// TIA Portal V17 export
// export: Created 2024-09-02T12:50:26.1404995Z, ExportSetting WithDefaults, DisplayName Totally Integrated Automation Portal, DisplayVersion V17, DisplayName TIA Portal Openness, DisplayVersion V17, DisplayName TIA Portal Version Control Interface, DisplayVersion V17, DisplayName STEP 7 Professional, DisplayVersion V17, DisplayName STEP 7 Safety, DisplayVersion V17, DisplayName WinCC Professional, DisplayVersion V17
TYPE "type_HMI_EKS_DATA"
// stored: IsFailsafeCompliant false
   STRUCT
      EKSAdapterIndex : UInt;
      CostCenter : Array[0..3] of Char;   // EKS Data Byte 84 - 87: Kostenstelle / EKS data bytes 84 - 87: cost center
      DateEnd : Array[0..7] of Char;   // EKS Data Byte 88 - 95: Ablaufdatum / EKS data bytes 88 - 95: expiry date
      ProtectionLevel : Int;   // Protection Level, Schutzstufe / Protection level, Schutzstufe
      Operator_ID : Array[1..7] of Char;   // EKS Data Byte 97 - 103: Werker ID / EKS data bytes 97 - 103: operator ID
      SafetyMode : Byte;   // EKS Data Byte 104: Sichere Betriebsart / EKS data byte 104: safe operating mode
      Specialbits : Byte;   // EKS Data Byte 105: Sonderbits / EKS data byte 105: special bits
      SerialNumber : Array[1..8] of Byte;   // EKS Data Byte 116 - 123: Seriennummer / EKS data bytes 116 - 123: serial number
      KeyAdapterReady : Bool;   // EKS Adapter betriebsbereit / EKS adapter ready
      KeyDetected : Bool;   // EKS Adapter Key erkannt / EKS adapter key detected
      ChecksumNotOK : Bool;   // Schlüsseldaten: Checksumme nicht in Ordnung / Key data: checksum not OK
      DateNotOK : Bool;   // Schlüsseldaten: Ablaufdatum überschritten / Key data: expiry date passed
      CostCenterNotOK : Bool;   // Schlüsseldaten: Kostenstelle nicht in Ordnung / Key data: cost center not OK
      KeyDataNotOK : Bool;   // Schlüsseldaten: Daten nicht in Ordnung / Key data: data not OK
      EKSKeyInvalidLess30Days : Bool;   // EKS Key invalid less than 30 days, EKS Schlüssel wird in weniger als 30 Tagen ungültig / EKS key invalid in less than 30 days, EKS Schlüssel wird in weniger als 30 Tagen ungültig
   END_STRUCT;
END_TYPE
